TYPE ST_Tank :
STRUCT
	 nId : INT;
     rtemperature : REAL;
     rlevel : REAL;
     bAlarm : BOOL ;
END_STRUCT
END_TYPE

(* stored: Version 1.1.0.1, ProductVersion 3.1.4024.16
   DUT ST_Tank: Id {7b8489ad-13ab-400c-82ec-922ac2567fd0} *)
